(* delete old files and delete oldest files if number of files exceeds specified number *)
PROGRAM C09_MaintainFolders_ORG
VAR
	tArchiveCheck				: TIME := t#4s;
	fbMaintainArchive			: FB_PulseGenerator;
	tDeleteTimeCheck			: TIME := t#20m;
	fbMaintainDeleteTime		: FB_PulseGenerator;
	(*tDeleteItemCheck			: TIME := t#4s;
	fbMaintainDeleteItem		: FB_PulseGenerator;*)
	nActivateBitWord			: DWORD; (* if index increase 32 bits it is necceasry to declar 64 bits var like LREAL;*)

	fbMaintainFolders			: ARRAY[1..25] OF NT_StartProcess;
	bTest	: BOOL;
	(*fbMoveOHMToArchive		: FB_OHM_MoveToArchive;*)
	(*fbMoveCACToArchive		: FB_CAC_MoveToArchive;*)
	fbMoveCHMToArchive		: FB_CHM_MoveToArchive;
	bZipCHMArchive			: BOOL;
	rtrigZipAfetrPassthrough		: R_TRIG;
	bManualZip					: BOOL;

	(*fbCompresOHMArchive		: NT_StartProcess;
	fbCompresCHMArchive		: NT_StartProcess;
	fbCompresPHMArchive		: NT_StartProcess;

	fbDeleteCHMNoLabel		: NT_StartProcess;*)

	fbRestoreTimer			: TON;
	fbRestoreOACFromCAC		: FB_CAC_RestoreOAC;
	nOCVFilesRestored			: UDINT;
	nOACFilesRestored			: UDINT;
	nCACFilesRestored			: UDINT;

	(*rtrigClearOCV				: R_TRIG;
	rtrigClearOCVError			: R_TRIG;
	rtrigClearOAC				: R_TRIG;
	rtrigClearOACError			: R_TRIG;

	fbClearOCVArchive			: FB_OCV_ClearArchive;
	fbClearOCVError			: FB_OCV_ClearArchive;
	fbClearOACArchive			: FB_OAC_ClearArchive;
	fbClearOACError			: FB_OAC_ClearArchive;

	rtrigClearOHM_FLG			: R_TRIG;
	rtrigClearCHM_FLG			: R_TRIG;

	fbClearOHM_FLG			: FB_OHM_ClearFLG;
	fbClearCHM_FLG			: FB_CHM_ClearFLG;
	btest : BOOL;*)

(********************************************************************************
		cBASE_FOLDER_ARR	: ARRAY[1..cSYSTEM_FOLDER_LIMIT] OF T_FolderName :=
			(*01*)'Bridge\',		(*02*)'Bridge\Archive\',		(*03*)'Bridge\Restore\',
			(*04*)'CAC\',		(*05*)'CAC\Archive\',		(*06*)'CAC\Error\',		(*07*)'CAC\Restore\', 	(*08*)'CAC\Restore\Archive\',
			(*09*)'CHM\',		(*10*)'CHM\Archive\',		(*11*)'CHM\Error\',		(*12*)'CHM\OK\',		(*13*)'CHM\Commissioning_Mode\',
			(*14*)'HMI\',
			(*15*)'KPI\',		(*16*)'KPI\Archive\',			(*17*)'KPI\Shift\',		(*18*)'KPI\ProdOrder\',
			(*19*)'OAC\',		(*20*)'OAC\Error\',
			(*21*)'OCV\',		(*22*)'OCV\Error\',
			(*23*)'OHM\',		(*24*)'OHM\Archive\',		(*25*)'OHM\Error\',		(*26*)'OHM\OK\',		(*27*)'OHM\Pending\',
			(*28*)'PCM\',		(*29*)'PCM\Archive\',		(*30*)'PCM\Error\',		(*31*)'PCM\Incoming\',
			(*32*)'PAC\',
			(*33*)'PHM\',		(*34*)'PHM\Archive\',		(*35*)'PHM\Error\',		(*36*)'PHM\OK\',
			(*37*)'Settings\',	(*38*)'Settings\Backups\',
			(*39*)'Templates\',
			(*40*)'Orca\',
			(*41*) 'SystemLog\';

*************************************************************************************)
END_VAR

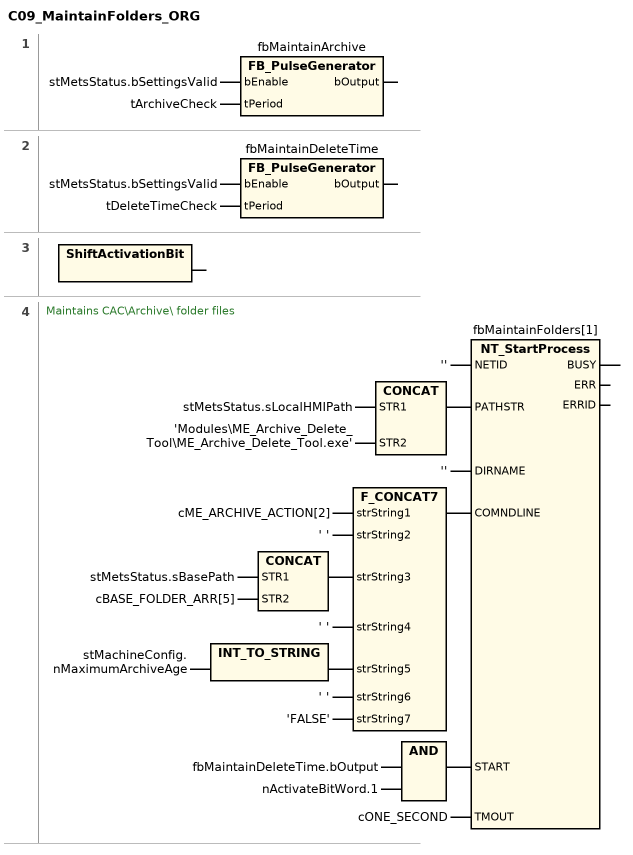
// NETWORK 1
fbMaintainArchive(bEnable := stMetsStatus.bSettingsValid, tPeriod := tArchiveCheck); // FB_PulseGenerator

// NETWORK 2
fbMaintainDeleteTime(bEnable := stMetsStatus.bSettingsValid, tPeriod := tDeleteTimeCheck); // FB_PulseGenerator

// NETWORK 3
ShiftActivationBit();

// NETWORK 4
// Maintains CAC\Archive\ folder files
fbMaintainFolders[1](
    NETID := '',
    PATHSTR := CONCAT(STR1 := stMetsStatus.sLocalHMIPath, STR2 := 'Modules\ME_Archive_Delete_Tool\ME_Archive_Delete_Tool.exe'),
    DIRNAME := '',
    COMNDLINE := F_CONCAT7(strString1 := cME_ARCHIVE_ACTION[2], strString2 := ' ', strString3 := CONCAT(STR1 := stMetsStatus.sBasePath, STR2 := cBASE_FOLDER_ARR[5]), strString4 := ' ', strString5 := INT_TO_STRING(stMachineConfig.nMaximumArchiveAge), strString6 := ' ', strString7 := 'FALSE'),
    START := fbMaintainDeleteTime.bOutput AND nActivateBitWord.1,
    TMOUT := cONE_SECOND); // NT_StartProcess

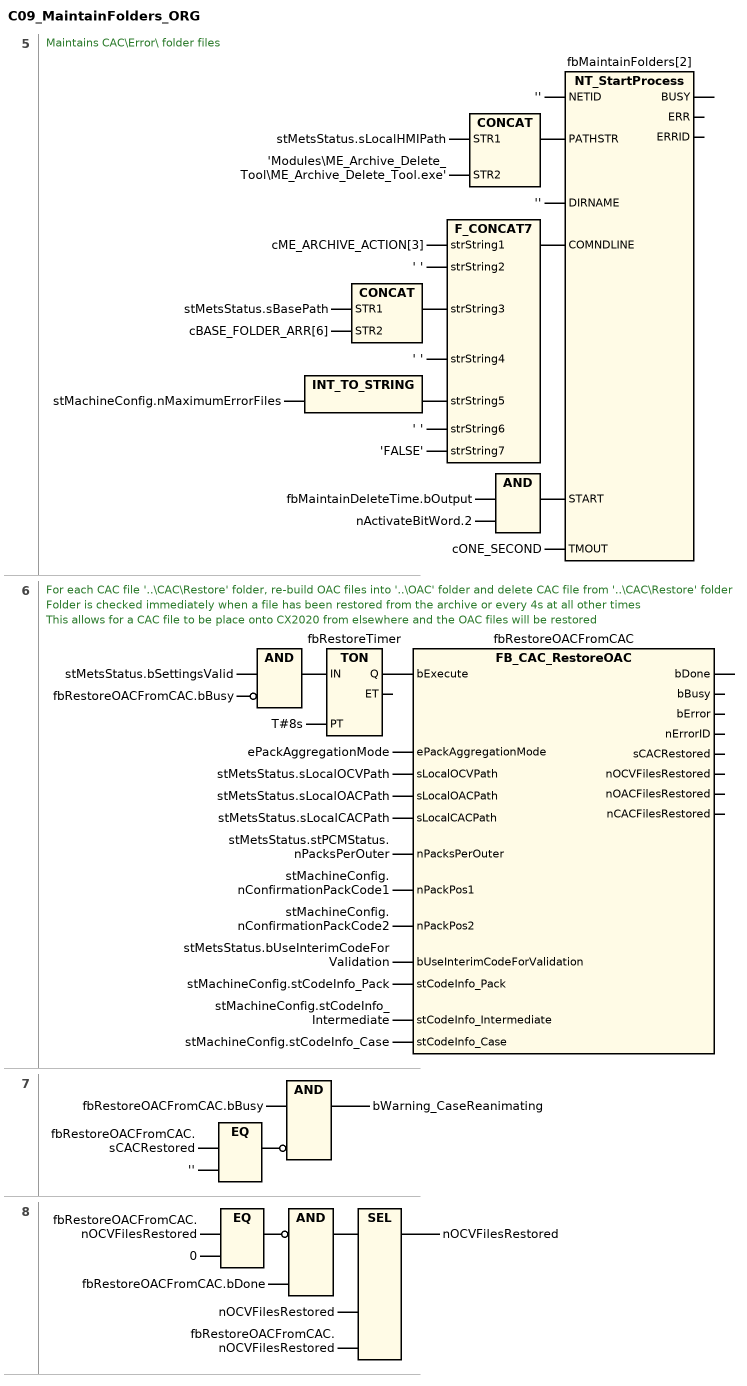
// NETWORK 5
// Maintains CAC\Error\ folder files
fbMaintainFolders[2](
    NETID := '',
    PATHSTR := CONCAT(STR1 := stMetsStatus.sLocalHMIPath, STR2 := 'Modules\ME_Archive_Delete_Tool\ME_Archive_Delete_Tool.exe'),
    DIRNAME := '',
    COMNDLINE := F_CONCAT7(strString1 := cME_ARCHIVE_ACTION[3], strString2 := ' ', strString3 := CONCAT(STR1 := stMetsStatus.sBasePath, STR2 := cBASE_FOLDER_ARR[6]), strString4 := ' ', strString5 := INT_TO_STRING(stMachineConfig.nMaximumErrorFiles), strString6 := ' ', strString7 := 'FALSE'),
    START := fbMaintainDeleteTime.bOutput AND nActivateBitWord.2,
    TMOUT := cONE_SECOND); // NT_StartProcess

// NETWORK 6
// 					For each CAC file '..\CAC\Restore' folder, re-build OAC files into '..\OAC' folder and delete CAC file from '..\CAC\Restore' folder
// Folder is checked immediately when a file has been restored from the archive or every 4s at all other times
// This allows for a CAC file to be place onto CX2020 from elsewhere and the OAC files will be restored
//
fbRestoreTimer(IN := stMetsStatus.bSettingsValid AND NOT fbRestoreOACFromCAC.bBusy, PT := T#8s); // TON
fbRestoreOACFromCAC(
    bExecute := fbRestoreTimer.Q,
    ePackAggregationMode := ePackAggregationMode,
    sLocalOCVPath := stMetsStatus.sLocalOCVPath,
    sLocalOACPath := stMetsStatus.sLocalOACPath,
    sLocalCACPath := stMetsStatus.sLocalCACPath,
    nPacksPerOuter := stMetsStatus.stPCMStatus.nPacksPerOuter,
    nPackPos1 := stMachineConfig.nConfirmationPackCode1,
    nPackPos2 := stMachineConfig.nConfirmationPackCode2,
    bUseInterimCodeForValidation := stMetsStatus.bUseInterimCodeForValidation,
    stCodeInfo_Pack := stMachineConfig.stCodeInfo_Pack,
    stCodeInfo_Intermediate := stMachineConfig.stCodeInfo_Intermediate,
    stCodeInfo_Case := stMachineConfig.stCodeInfo_Case); // FB_CAC_RestoreOAC

// NETWORK 7
bWarning_CaseReanimating := fbRestoreOACFromCAC.bBusy AND NOT (fbRestoreOACFromCAC.sCACRestored = '');

// NETWORK 8
nOCVFilesRestored := SEL(NOT (fbRestoreOACFromCAC.nOCVFilesRestored = 0) AND fbRestoreOACFromCAC.bDone, nOCVFilesRestored, fbRestoreOACFromCAC.nOCVFilesRestored);

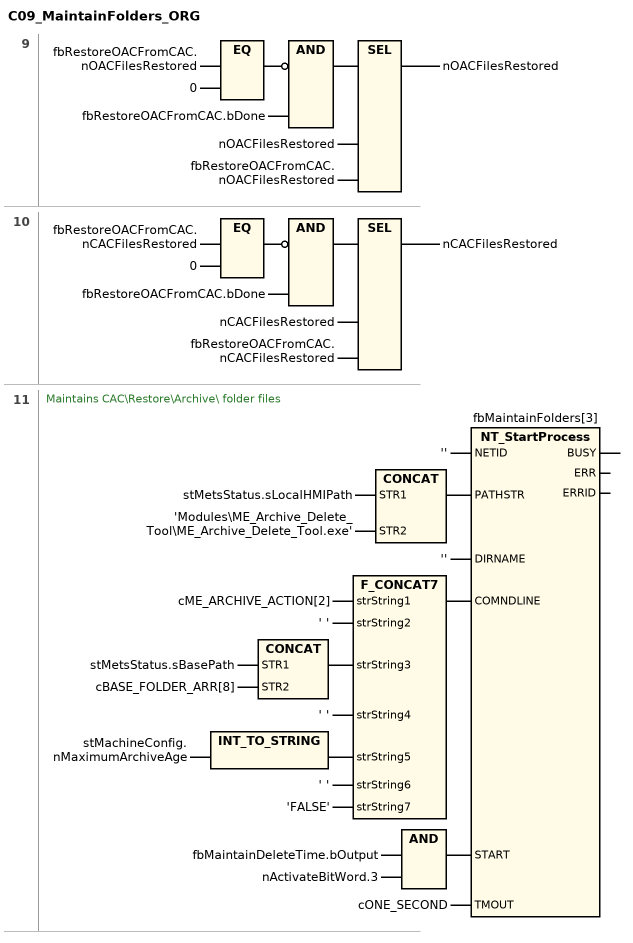
// NETWORK 9
nOACFilesRestored := SEL(NOT (fbRestoreOACFromCAC.nOACFilesRestored = 0) AND fbRestoreOACFromCAC.bDone, nOACFilesRestored, fbRestoreOACFromCAC.nOACFilesRestored);

// NETWORK 10
nCACFilesRestored := SEL(NOT (fbRestoreOACFromCAC.nCACFilesRestored = 0) AND fbRestoreOACFromCAC.bDone, nCACFilesRestored, fbRestoreOACFromCAC.nCACFilesRestored);

// NETWORK 11
// Maintains CAC\Restore\Archive\ folder files
fbMaintainFolders[3](
    NETID := '',
    PATHSTR := CONCAT(STR1 := stMetsStatus.sLocalHMIPath, STR2 := 'Modules\ME_Archive_Delete_Tool\ME_Archive_Delete_Tool.exe'),
    DIRNAME := '',
    COMNDLINE := F_CONCAT7(strString1 := cME_ARCHIVE_ACTION[2], strString2 := ' ', strString3 := CONCAT(STR1 := stMetsStatus.sBasePath, STR2 := cBASE_FOLDER_ARR[8]), strString4 := ' ', strString5 := INT_TO_STRING(stMachineConfig.nMaximumArchiveAge), strString6 := ' ', strString7 := 'FALSE'),
    START := fbMaintainDeleteTime.bOutput AND nActivateBitWord.3,
    TMOUT := cONE_SECOND); // NT_StartProcess

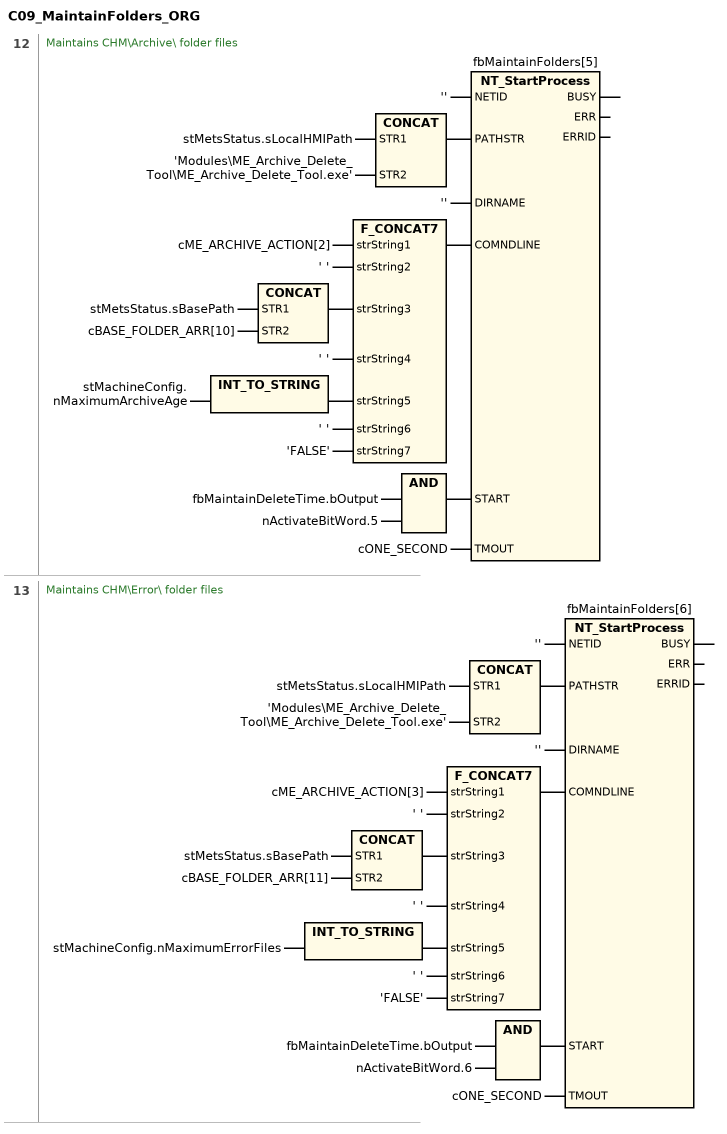
// NETWORK 12
// Maintains CHM\Archive\ folder files
fbMaintainFolders[5](
    NETID := '',
    PATHSTR := CONCAT(STR1 := stMetsStatus.sLocalHMIPath, STR2 := 'Modules\ME_Archive_Delete_Tool\ME_Archive_Delete_Tool.exe'),
    DIRNAME := '',
    COMNDLINE := F_CONCAT7(strString1 := cME_ARCHIVE_ACTION[2], strString2 := ' ', strString3 := CONCAT(STR1 := stMetsStatus.sBasePath, STR2 := cBASE_FOLDER_ARR[10]), strString4 := ' ', strString5 := INT_TO_STRING(stMachineConfig.nMaximumArchiveAge), strString6 := ' ', strString7 := 'FALSE'),
    START := fbMaintainDeleteTime.bOutput AND nActivateBitWord.5,
    TMOUT := cONE_SECOND); // NT_StartProcess

// NETWORK 13
// Maintains CHM\Error\ folder files
fbMaintainFolders[6](
    NETID := '',
    PATHSTR := CONCAT(STR1 := stMetsStatus.sLocalHMIPath, STR2 := 'Modules\ME_Archive_Delete_Tool\ME_Archive_Delete_Tool.exe'),
    DIRNAME := '',
    COMNDLINE := F_CONCAT7(strString1 := cME_ARCHIVE_ACTION[3], strString2 := ' ', strString3 := CONCAT(STR1 := stMetsStatus.sBasePath, STR2 := cBASE_FOLDER_ARR[11]), strString4 := ' ', strString5 := INT_TO_STRING(stMachineConfig.nMaximumErrorFiles), strString6 := ' ', strString7 := 'FALSE'),
    START := fbMaintainDeleteTime.bOutput AND nActivateBitWord.6,
    TMOUT := cONE_SECOND); // NT_StartProcess

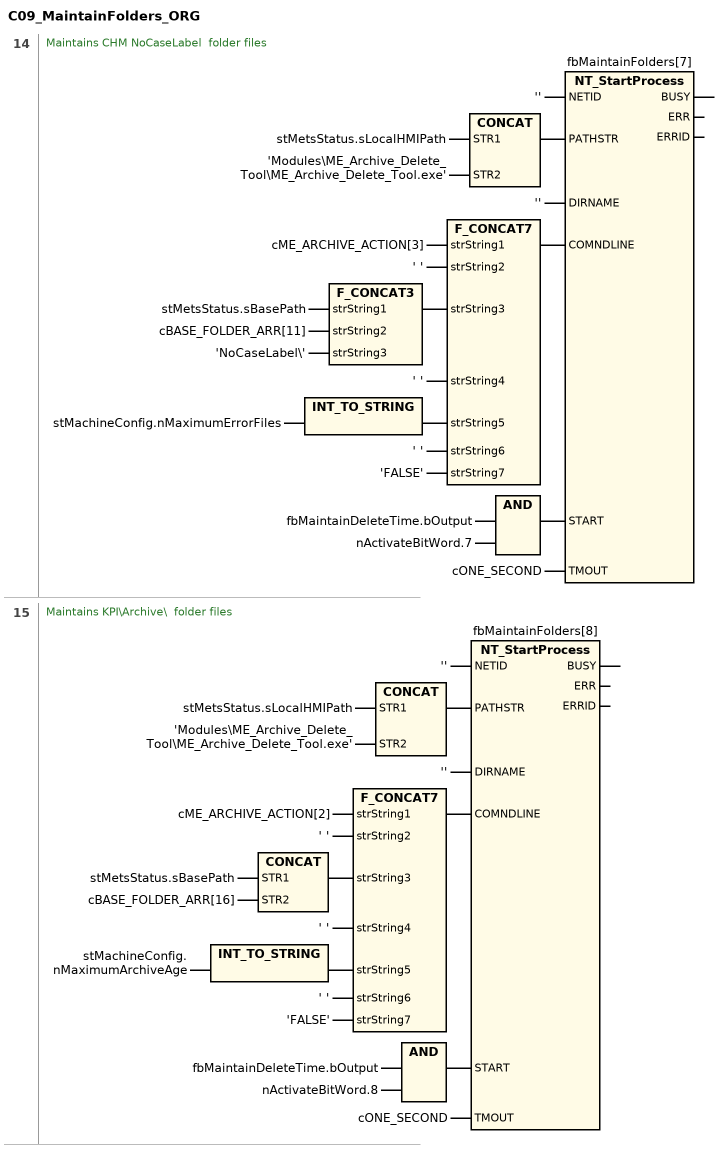
// NETWORK 14
// Maintains CHM NoCaseLabel  folder files
fbMaintainFolders[7](
    NETID := '',
    PATHSTR := CONCAT(STR1 := stMetsStatus.sLocalHMIPath, STR2 := 'Modules\ME_Archive_Delete_Tool\ME_Archive_Delete_Tool.exe'),
    DIRNAME := '',
    COMNDLINE := F_CONCAT7(strString1 := cME_ARCHIVE_ACTION[3], strString2 := ' ', strString3 := F_CONCAT3(strString1 := stMetsStatus.sBasePath, strString2 := cBASE_FOLDER_ARR[11], strString3 := 'NoCaseLabel\'), strString4 := ' ', strString5 := INT_TO_STRING(stMachineConfig.nMaximumErrorFiles), strString6 := ' ', strString7 := 'FALSE'),
    START := fbMaintainDeleteTime.bOutput AND nActivateBitWord.7,
    TMOUT := cONE_SECOND); // NT_StartProcess

// NETWORK 15
// Maintains KPI\Archive\  folder files
fbMaintainFolders[8](
    NETID := '',
    PATHSTR := CONCAT(STR1 := stMetsStatus.sLocalHMIPath, STR2 := 'Modules\ME_Archive_Delete_Tool\ME_Archive_Delete_Tool.exe'),
    DIRNAME := '',
    COMNDLINE := F_CONCAT7(strString1 := cME_ARCHIVE_ACTION[2], strString2 := ' ', strString3 := CONCAT(STR1 := stMetsStatus.sBasePath, STR2 := cBASE_FOLDER_ARR[16]), strString4 := ' ', strString5 := INT_TO_STRING(stMachineConfig.nMaximumArchiveAge), strString6 := ' ', strString7 := 'FALSE'),
    START := fbMaintainDeleteTime.bOutput AND nActivateBitWord.8,
    TMOUT := cONE_SECOND); // NT_StartProcess

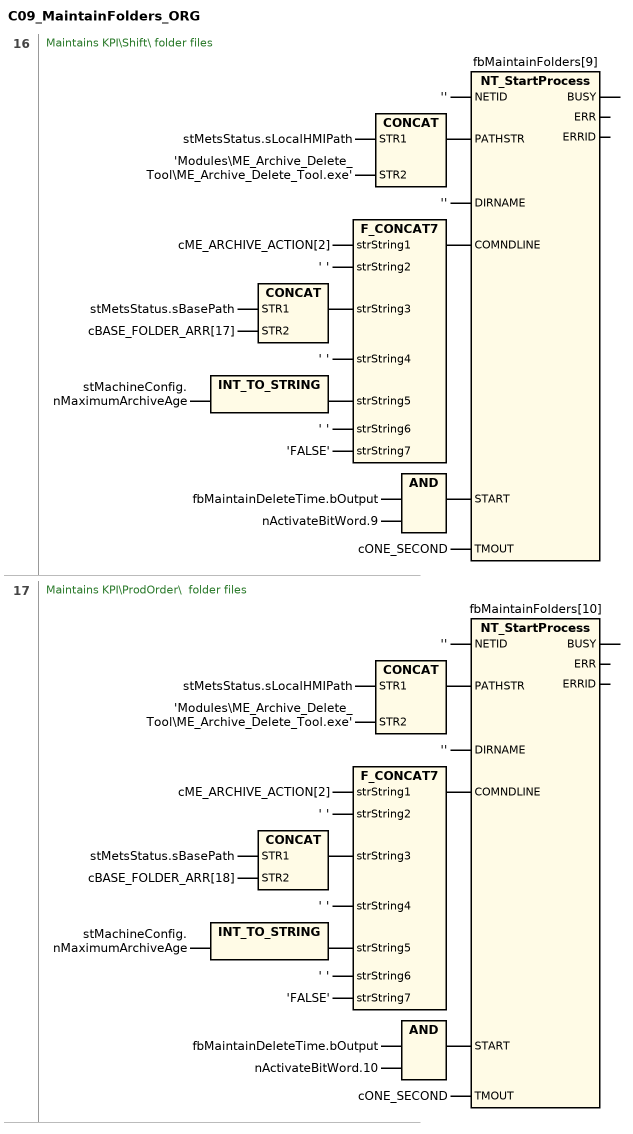
// NETWORK 16
// Maintains KPI\Shift\ folder files
fbMaintainFolders[9](
    NETID := '',
    PATHSTR := CONCAT(STR1 := stMetsStatus.sLocalHMIPath, STR2 := 'Modules\ME_Archive_Delete_Tool\ME_Archive_Delete_Tool.exe'),
    DIRNAME := '',
    COMNDLINE := F_CONCAT7(strString1 := cME_ARCHIVE_ACTION[2], strString2 := ' ', strString3 := CONCAT(STR1 := stMetsStatus.sBasePath, STR2 := cBASE_FOLDER_ARR[17]), strString4 := ' ', strString5 := INT_TO_STRING(stMachineConfig.nMaximumArchiveAge), strString6 := ' ', strString7 := 'FALSE'),
    START := fbMaintainDeleteTime.bOutput AND nActivateBitWord.9,
    TMOUT := cONE_SECOND); // NT_StartProcess

// NETWORK 17
// Maintains KPI\ProdOrder\  folder files
fbMaintainFolders[10](
    NETID := '',
    PATHSTR := CONCAT(STR1 := stMetsStatus.sLocalHMIPath, STR2 := 'Modules\ME_Archive_Delete_Tool\ME_Archive_Delete_Tool.exe'),
    DIRNAME := '',
    COMNDLINE := F_CONCAT7(strString1 := cME_ARCHIVE_ACTION[2], strString2 := ' ', strString3 := CONCAT(STR1 := stMetsStatus.sBasePath, STR2 := cBASE_FOLDER_ARR[18]), strString4 := ' ', strString5 := INT_TO_STRING(stMachineConfig.nMaximumArchiveAge), strString6 := ' ', strString7 := 'FALSE'),
    START := fbMaintainDeleteTime.bOutput AND nActivateBitWord.10,
    TMOUT := cONE_SECOND); // NT_StartProcess

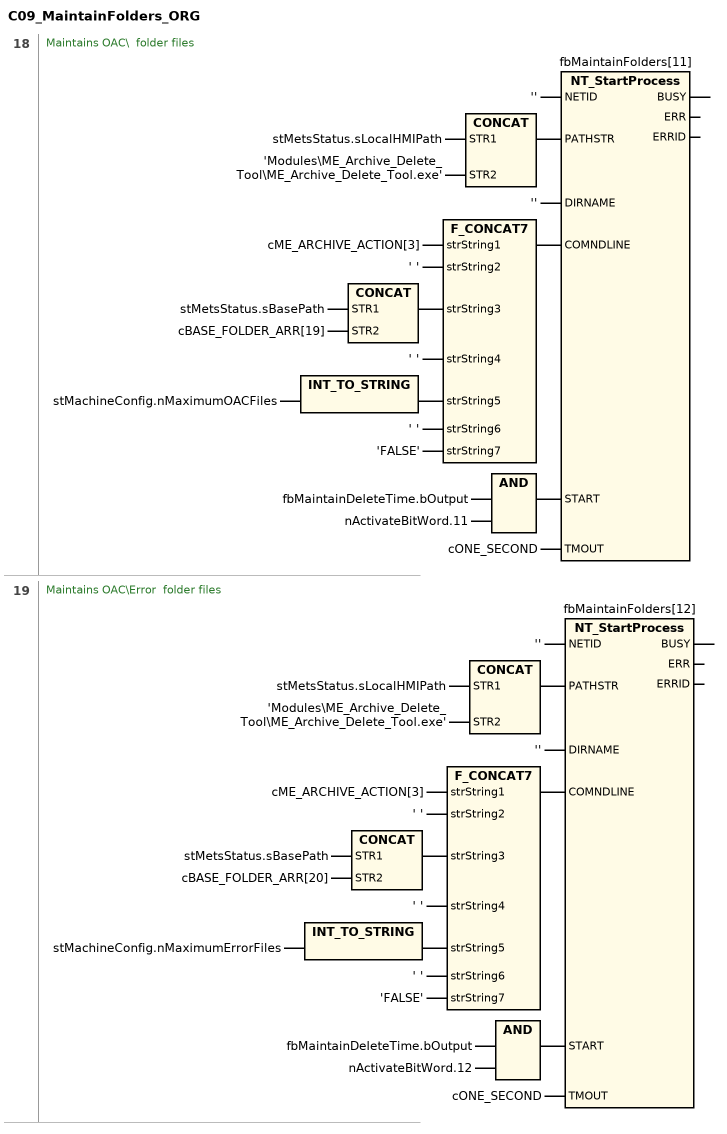
// NETWORK 18
// Maintains OAC\  folder files
fbMaintainFolders[11](
    NETID := '',
    PATHSTR := CONCAT(STR1 := stMetsStatus.sLocalHMIPath, STR2 := 'Modules\ME_Archive_Delete_Tool\ME_Archive_Delete_Tool.exe'),
    DIRNAME := '',
    COMNDLINE := F_CONCAT7(strString1 := cME_ARCHIVE_ACTION[3], strString2 := ' ', strString3 := CONCAT(STR1 := stMetsStatus.sBasePath, STR2 := cBASE_FOLDER_ARR[19]), strString4 := ' ', strString5 := INT_TO_STRING(stMachineConfig.nMaximumOACFiles), strString6 := ' ', strString7 := 'FALSE'),
    START := fbMaintainDeleteTime.bOutput AND nActivateBitWord.11,
    TMOUT := cONE_SECOND); // NT_StartProcess

// NETWORK 19
// Maintains OAC\Error  folder files
fbMaintainFolders[12](
    NETID := '',
    PATHSTR := CONCAT(STR1 := stMetsStatus.sLocalHMIPath, STR2 := 'Modules\ME_Archive_Delete_Tool\ME_Archive_Delete_Tool.exe'),
    DIRNAME := '',
    COMNDLINE := F_CONCAT7(strString1 := cME_ARCHIVE_ACTION[3], strString2 := ' ', strString3 := CONCAT(STR1 := stMetsStatus.sBasePath, STR2 := cBASE_FOLDER_ARR[20]), strString4 := ' ', strString5 := INT_TO_STRING(stMachineConfig.nMaximumErrorFiles), strString6 := ' ', strString7 := 'FALSE'),
    START := fbMaintainDeleteTime.bOutput AND nActivateBitWord.12,
    TMOUT := cONE_SECOND); // NT_StartProcess

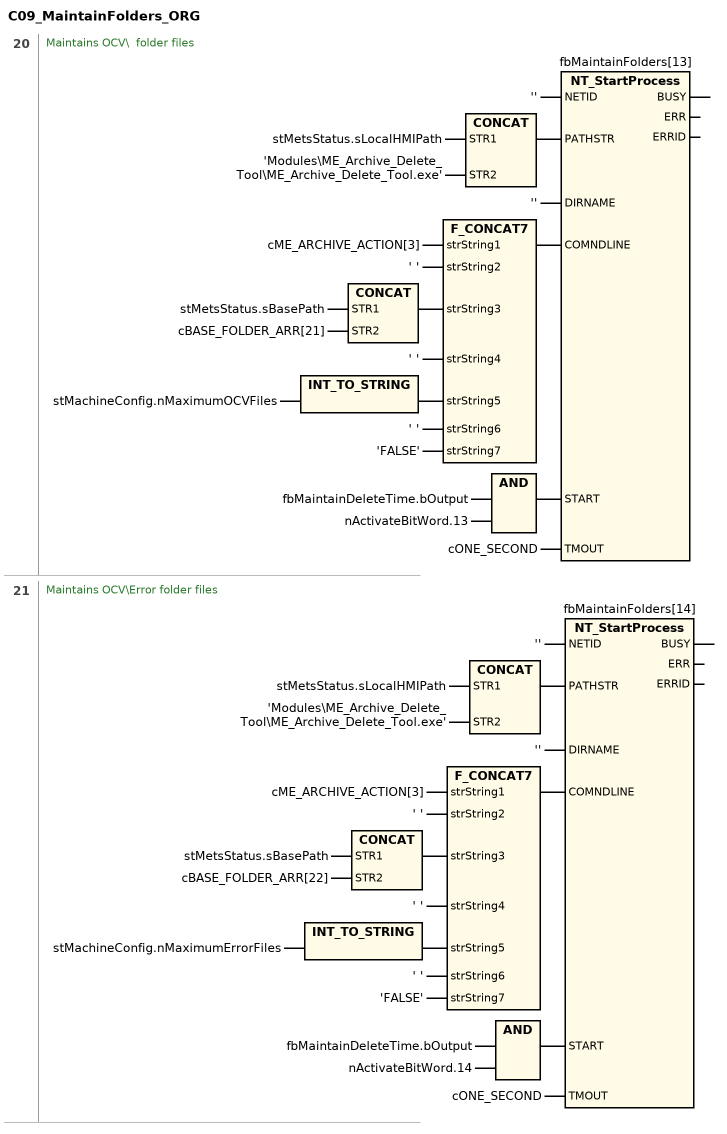
// NETWORK 20
// Maintains OCV\  folder files
fbMaintainFolders[13](
    NETID := '',
    PATHSTR := CONCAT(STR1 := stMetsStatus.sLocalHMIPath, STR2 := 'Modules\ME_Archive_Delete_Tool\ME_Archive_Delete_Tool.exe'),
    DIRNAME := '',
    COMNDLINE := F_CONCAT7(strString1 := cME_ARCHIVE_ACTION[3], strString2 := ' ', strString3 := CONCAT(STR1 := stMetsStatus.sBasePath, STR2 := cBASE_FOLDER_ARR[21]), strString4 := ' ', strString5 := INT_TO_STRING(stMachineConfig.nMaximumOCVFiles), strString6 := ' ', strString7 := 'FALSE'),
    START := fbMaintainDeleteTime.bOutput AND nActivateBitWord.13,
    TMOUT := cONE_SECOND); // NT_StartProcess

// NETWORK 21
// Maintains OCV\Error folder files
fbMaintainFolders[14](
    NETID := '',
    PATHSTR := CONCAT(STR1 := stMetsStatus.sLocalHMIPath, STR2 := 'Modules\ME_Archive_Delete_Tool\ME_Archive_Delete_Tool.exe'),
    DIRNAME := '',
    COMNDLINE := F_CONCAT7(strString1 := cME_ARCHIVE_ACTION[3], strString2 := ' ', strString3 := CONCAT(STR1 := stMetsStatus.sBasePath, STR2 := cBASE_FOLDER_ARR[22]), strString4 := ' ', strString5 := INT_TO_STRING(stMachineConfig.nMaximumErrorFiles), strString6 := ' ', strString7 := 'FALSE'),
    START := fbMaintainDeleteTime.bOutput AND nActivateBitWord.14,
    TMOUT := cONE_SECOND); // NT_StartProcess

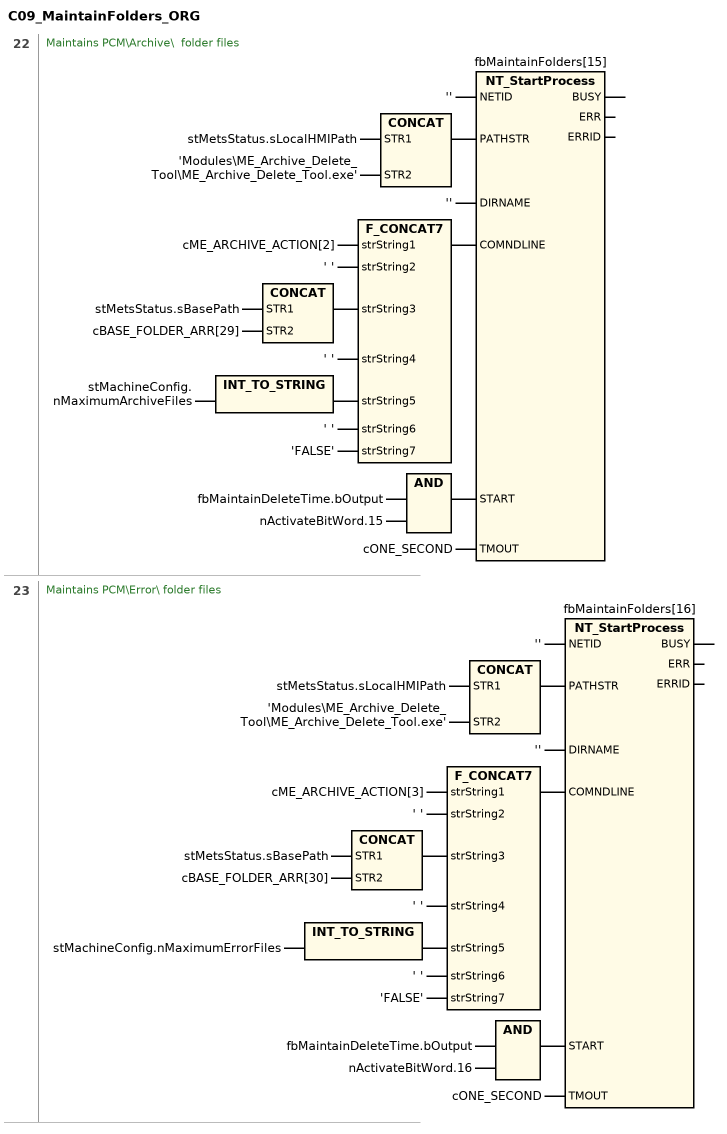
// NETWORK 22
// Maintains PCM\Archive\  folder files
fbMaintainFolders[15](
    NETID := '',
    PATHSTR := CONCAT(STR1 := stMetsStatus.sLocalHMIPath, STR2 := 'Modules\ME_Archive_Delete_Tool\ME_Archive_Delete_Tool.exe'),
    DIRNAME := '',
    COMNDLINE := F_CONCAT7(strString1 := cME_ARCHIVE_ACTION[2], strString2 := ' ', strString3 := CONCAT(STR1 := stMetsStatus.sBasePath, STR2 := cBASE_FOLDER_ARR[29]), strString4 := ' ', strString5 := INT_TO_STRING(stMachineConfig.nMaximumArchiveFiles), strString6 := ' ', strString7 := 'FALSE'),
    START := fbMaintainDeleteTime.bOutput AND nActivateBitWord.15,
    TMOUT := cONE_SECOND); // NT_StartProcess

// NETWORK 23
// Maintains PCM\Error\ folder files
fbMaintainFolders[16](
    NETID := '',
    PATHSTR := CONCAT(STR1 := stMetsStatus.sLocalHMIPath, STR2 := 'Modules\ME_Archive_Delete_Tool\ME_Archive_Delete_Tool.exe'),
    DIRNAME := '',
    COMNDLINE := F_CONCAT7(strString1 := cME_ARCHIVE_ACTION[3], strString2 := ' ', strString3 := CONCAT(STR1 := stMetsStatus.sBasePath, STR2 := cBASE_FOLDER_ARR[30]), strString4 := ' ', strString5 := INT_TO_STRING(stMachineConfig.nMaximumErrorFiles), strString6 := ' ', strString7 := 'FALSE'),
    START := fbMaintainDeleteTime.bOutput AND nActivateBitWord.16,
    TMOUT := cONE_SECOND); // NT_StartProcess

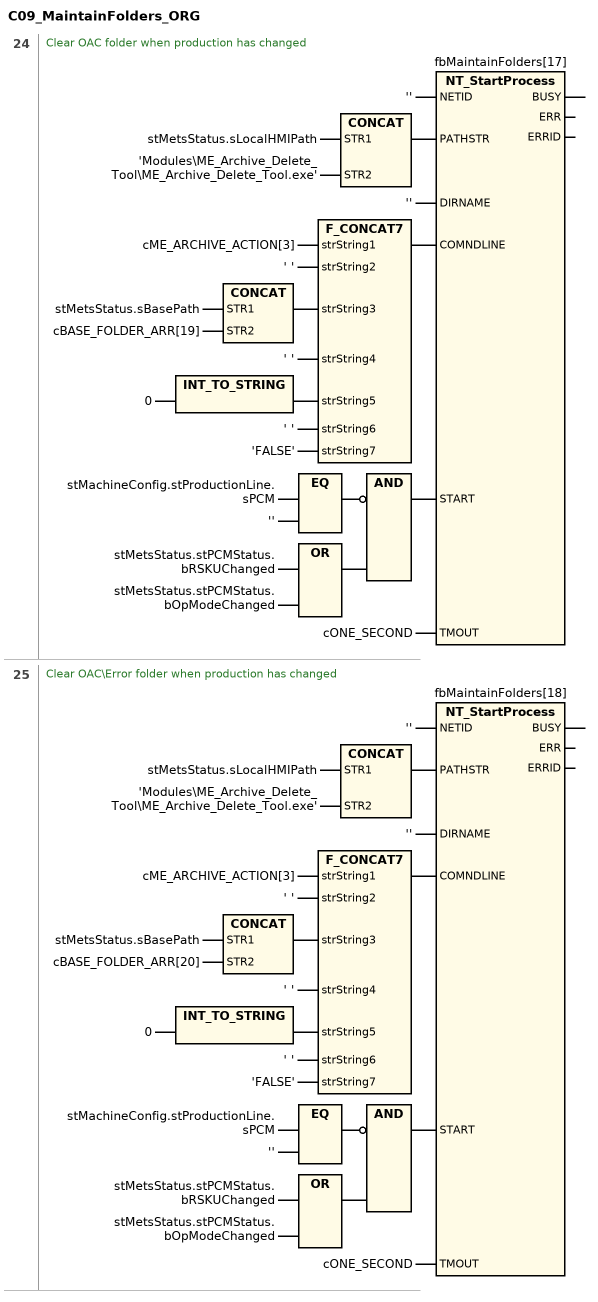
// NETWORK 24
// Clear OAC folder when production has changed
fbMaintainFolders[17](
    NETID := '',
    PATHSTR := CONCAT(STR1 := stMetsStatus.sLocalHMIPath, STR2 := 'Modules\ME_Archive_Delete_Tool\ME_Archive_Delete_Tool.exe'),
    DIRNAME := '',
    COMNDLINE := F_CONCAT7(strString1 := cME_ARCHIVE_ACTION[3], strString2 := ' ', strString3 := CONCAT(STR1 := stMetsStatus.sBasePath, STR2 := cBASE_FOLDER_ARR[19]), strString4 := ' ', strString5 := INT_TO_STRING(0), strString6 := ' ', strString7 := 'FALSE'),
    START := NOT (stMachineConfig.stProductionLine.sPCM = '') AND (stMetsStatus.stPCMStatus.bRSKUChanged OR stMetsStatus.stPCMStatus.bOpModeChanged),
    TMOUT := cONE_SECOND); // NT_StartProcess

// NETWORK 25
// Clear OAC\Error folder when production has changed
fbMaintainFolders[18](
    NETID := '',
    PATHSTR := CONCAT(STR1 := stMetsStatus.sLocalHMIPath, STR2 := 'Modules\ME_Archive_Delete_Tool\ME_Archive_Delete_Tool.exe'),
    DIRNAME := '',
    COMNDLINE := F_CONCAT7(strString1 := cME_ARCHIVE_ACTION[3], strString2 := ' ', strString3 := CONCAT(STR1 := stMetsStatus.sBasePath, STR2 := cBASE_FOLDER_ARR[20]), strString4 := ' ', strString5 := INT_TO_STRING(0), strString6 := ' ', strString7 := 'FALSE'),
    START := NOT (stMachineConfig.stProductionLine.sPCM = '') AND (stMetsStatus.stPCMStatus.bRSKUChanged OR stMetsStatus.stPCMStatus.bOpModeChanged),
    TMOUT := cONE_SECOND); // NT_StartProcess

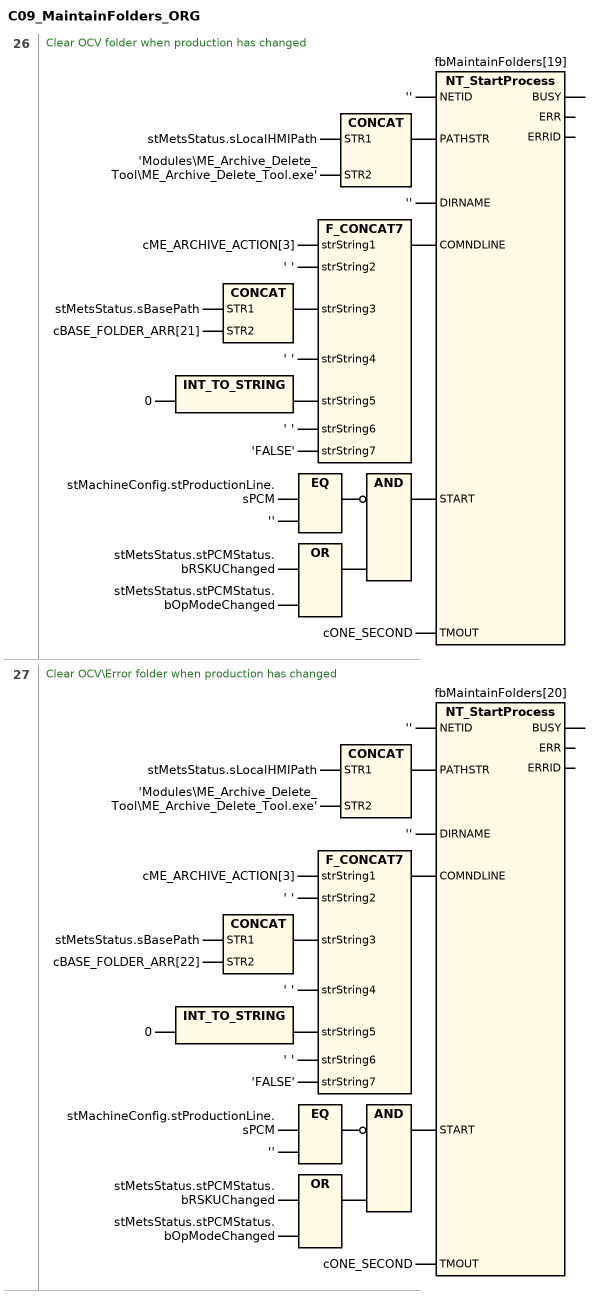
// NETWORK 26
// Clear OCV folder when production has changed
fbMaintainFolders[19](
    NETID := '',
    PATHSTR := CONCAT(STR1 := stMetsStatus.sLocalHMIPath, STR2 := 'Modules\ME_Archive_Delete_Tool\ME_Archive_Delete_Tool.exe'),
    DIRNAME := '',
    COMNDLINE := F_CONCAT7(strString1 := cME_ARCHIVE_ACTION[3], strString2 := ' ', strString3 := CONCAT(STR1 := stMetsStatus.sBasePath, STR2 := cBASE_FOLDER_ARR[21]), strString4 := ' ', strString5 := INT_TO_STRING(0), strString6 := ' ', strString7 := 'FALSE'),
    START := NOT (stMachineConfig.stProductionLine.sPCM = '') AND (stMetsStatus.stPCMStatus.bRSKUChanged OR stMetsStatus.stPCMStatus.bOpModeChanged),
    TMOUT := cONE_SECOND); // NT_StartProcess

// NETWORK 27
// Clear OCV\Error folder when production has changed
fbMaintainFolders[20](
    NETID := '',
    PATHSTR := CONCAT(STR1 := stMetsStatus.sLocalHMIPath, STR2 := 'Modules\ME_Archive_Delete_Tool\ME_Archive_Delete_Tool.exe'),
    DIRNAME := '',
    COMNDLINE := F_CONCAT7(strString1 := cME_ARCHIVE_ACTION[3], strString2 := ' ', strString3 := CONCAT(STR1 := stMetsStatus.sBasePath, STR2 := cBASE_FOLDER_ARR[22]), strString4 := ' ', strString5 := INT_TO_STRING(0), strString6 := ' ', strString7 := 'FALSE'),
    START := NOT (stMachineConfig.stProductionLine.sPCM = '') AND (stMetsStatus.stPCMStatus.bRSKUChanged OR stMetsStatus.stPCMStatus.bOpModeChanged),
    TMOUT := cONE_SECOND); // NT_StartProcess

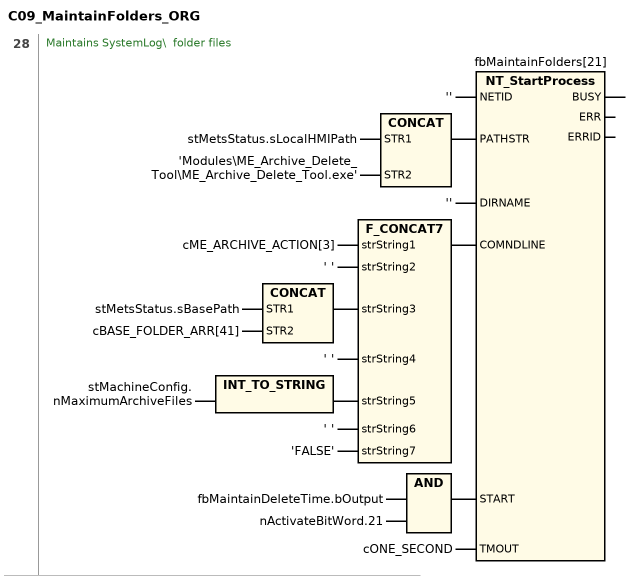
// NETWORK 28
// Maintains SystemLog\  folder files
fbMaintainFolders[21](
    NETID := '',
    PATHSTR := CONCAT(STR1 := stMetsStatus.sLocalHMIPath, STR2 := 'Modules\ME_Archive_Delete_Tool\ME_Archive_Delete_Tool.exe'),
    DIRNAME := '',
    COMNDLINE := F_CONCAT7(strString1 := cME_ARCHIVE_ACTION[3], strString2 := ' ', strString3 := CONCAT(STR1 := stMetsStatus.sBasePath, STR2 := cBASE_FOLDER_ARR[41]), strString4 := ' ', strString5 := INT_TO_STRING(stMachineConfig.nMaximumArchiveFiles), strString6 := ' ', strString7 := 'FALSE'),
    START := fbMaintainDeleteTime.bOutput AND nActivateBitWord.21,
    TMOUT := cONE_SECOND); // NT_StartProcess

ACTION ShiftActivationBit:
IF fbMaintainDeleteTime.bOutput	THEN
	IF nActivateBitWord = 0 THEN
		nActivateBitWord := 1;
	ELSE
		nActivateBitWord :=SHL(nActivateBitWord,1);
	END_IF
END_IF
END_ACTION

END_PROGRAM

(* stored: Version 1.1.0.1, ProductVersion 3.1.4024.15
   POU C09_MaintainFolders_ORG: Id {88f5b35a-c517-4510-82f2-39e07268058f}, SpecialFunc None
   Action ShiftActivationBit: Id {9e0a5311-b3b3-4fb0-a68b-309677878966} *)
